// Code généré automatiquement : NE PAS MODIFIER
FUNCTION CheckLRangeSigned : LINT
VAR_INPUT
	value, lower, upper: LINT;
END_VAR

// Code généré automatiquement : Il s’agit d’une proposition d’implémentation.
{noflow}
IF (value < lower) THEN
	CheckLRangeSigned := lower;
ELSIF(value > upper) THEN
	CheckLRangeSigned := upper;
ELSE
	CheckLRangeSigned := value;
END_IF

{flow}

END_FUNCTION

(* stored: Version 1.1.0.1, ProductVersion 3.1.4024.6
   POU CheckLRangeSigned: Id {a249d7fc-edec-4cbc-99e9-ea69de842367}, SpecialFunc CheckLRangeSigned *)
